FUNCTION_BLOCK old
VAR_INPUT
END_VAR
VAR_OUTPUT
END_VAR
VAR
END_VAR

ACTION BMSInit:
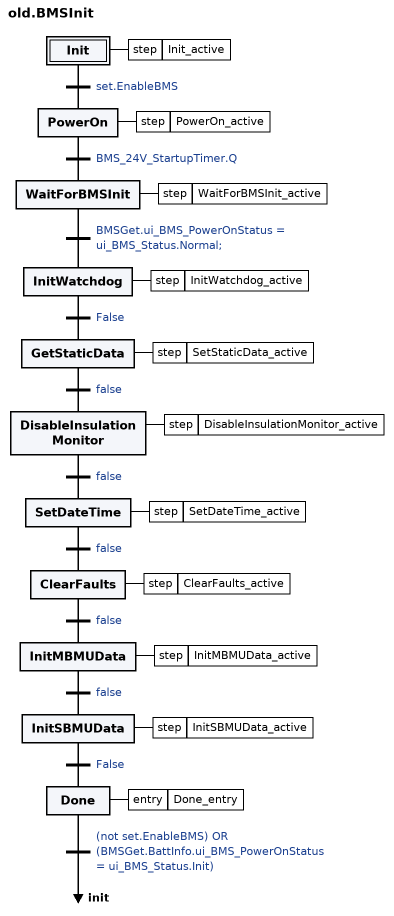
INITIAL_STEP Init:
    Init_active(N);  // step action
END_STEP
TRANSITION FROM Init TO PowerOn
    := set.EnableBMS;
END_TRANSITION
STEP PowerOn:
    PowerOn_active(N);  // step action
END_STEP
TRANSITION FROM PowerOn TO WaitForBMSInit
    := BMS_24V_StartupTimer.Q;
END_TRANSITION
STEP WaitForBMSInit:
    WaitForBMSInit_active(N);  // step action
END_STEP
TRANSITION FROM WaitForBMSInit TO InitWatchdog
    := BMSGet.ui_BMS_PowerOnStatus = ui_BMS_Status.Normal;
END_TRANSITION
STEP InitWatchdog:
    InitWatchdog_active(N);  // step action
END_STEP
TRANSITION FROM InitWatchdog TO GetStaticData
    := False;
END_TRANSITION
STEP GetStaticData:
    SetStaticData_active(N);  // step action
END_STEP
TRANSITION FROM GetStaticData TO DisableInsulationMonitor
    := false;
END_TRANSITION
STEP DisableInsulationMonitor:
    DisableInsulationMonitor_active(N);  // step action
END_STEP
TRANSITION FROM DisableInsulationMonitor TO SetDateTime
    := false;
END_TRANSITION
STEP SetDateTime:
    SetDateTime_active(N);  // step action
END_STEP
TRANSITION FROM SetDateTime TO ClearFaults
    := false;
END_TRANSITION
STEP ClearFaults:
    ClearFaults_active(N);  // step action
END_STEP
TRANSITION FROM ClearFaults TO InitMBMUData
    := false;
END_TRANSITION
STEP InitMBMUData:
    InitMBMUData_active(N);  // step action
END_STEP
TRANSITION FROM InitMBMUData TO InitSBMUData
    := false;
END_TRANSITION
STEP InitSBMUData:
    InitSBMUData_active(N);  // step action
END_STEP
TRANSITION FROM InitSBMUData TO Done
    := False;
END_TRANSITION
STEP Done:
    Done_entry(P1);  // entry action
END_STEP
TRANSITION FROM Done TO init
    := (not set.EnableBMS) OR (BMSGet.BattInfo.ui_BMS_PowerOnStatus = ui_BMS_Status.Init);
END_TRANSITION
END_ACTION

END_FUNCTION_BLOCK

(* stored: Version 1.1.0.1, ProductVersion 3.1.4024.12
   POU old: Id {b768a1b0-7b87-4091-b317-a71ef55e6617}, SpecialFunc None
   Action BMSInit: Id {15c0477e-db93-4291-b7cd-6c66ec1937f4} *)
